{attribute 'TcGenerated'}
{attribute 'no-analysis'}
{attribute 'linkalways'}
// This function has been automatically generated from the project information.
VAR_GLOBAL CONSTANT
	{attribute 'const_non_replaced'}
	stLibVersion_Library_Project : ST_LibVersion := (iMajor := 1, iMinor := 0, iBuild := 0, iRevision := 1, nFlags := 0, sVersion := '1.0.0.1');
END_VAR

(* stored: Version 1.1.0.1, ProductVersion 3.1.4024.14
   GVL Global_Version: Id {7062acdc-2a66-4515-aa94-1900bde78a80} *)
